Staubli VAL3: iPlate1.pgx

public program iPlate1(num& nNum[] (dimensions=1))
begin
  nNum=dioGet(iPlate1)
end
